// Mitsubishi GX Works2 project: tidal   PLC: FX3U/FX3UC

PROGRAM MAIN
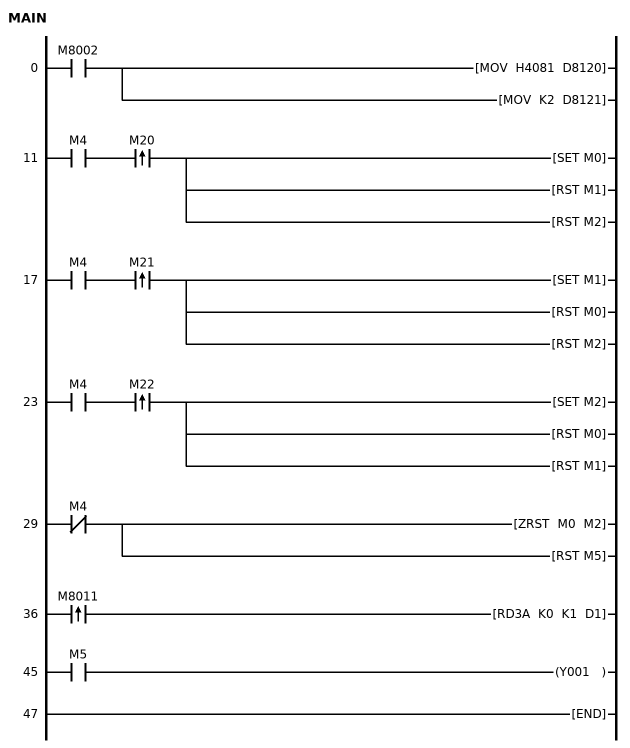
0     LD      M8002
      MOV     H4081 D8120
      MOV     K2 D8121
11    LD      M4
      ANDP    M20
      SET     M0
      RST     M1
      RST     M2
17    LD      M4
      ANDP    M21
      SET     M1
      RST     M0
      RST     M2
23    LD      M4
      ANDP    M22
      SET     M2
      RST     M0
      RST     M1
29    LDI     M4
      ZRST    M0 M2
      RST     M5
36    LDP     M8011
      RD3A    K0 K1 D1
45    LD      M5
      OUT     Y001
47    END
END_PROGRAM
